FUNCTION_BLOCK NE_BYTE (* IEC 61131-3 BYTE inequality test *)
  (* Standard: 61131-3 *)
  (* Version 0.0, 2006-09-14, JHC, Holobloc Inc *)
  (* Compiler header: package fb.rt.plc.bits; *)
  (* Compiler classdef: (IN1 != IN2) *)
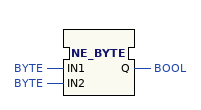
  VAR_INPUT
    IN1 : BYTE;
    IN2 : BYTE;
  END_VAR
  VAR_OUTPUT
    Q : BOOL;
  END_VAR
END_FUNCTION_BLOCK
